PROGRAM MAIN
VAR
	
	X	:	INT;

END_VAR

END_PROGRAM

(* stored: Version 1.1.0.1, ProductVersion 3.1.4024.3
   POU MAIN: Id {1fdbcb72-de71-4592-a01d-5e0a06697876}, SpecialFunc None *)
